// TIA Portal V19 program export: 4 tag tables, 0 data types, 0 data blocks, 1 code blocks (in call order from the OBs), 0 instance data blocks

VAR_GLOBAL   // PLC tag table "conveyor-0"
   "Start Button 0" AT %I0.0 : Bool;
   "Belt Conveyor (4m) 0" AT %Q0.0 : Bool;
   "memedge0-0" AT %M0.0 : Bool;
   "memedge0-1" AT %M0.1 : Bool;
   "memedge0-2" AT %M0.2 : Bool;
   "mem0-start" AT %M0.3 : Bool;
   "memory0-0" AT %M0.4 : Bool;
   "memedge0-3" AT %M0.5 : Bool;
   "memedge0-4" AT %M0.6 : Bool;
   "memedge0-5" AT %M0.7 : Bool;
END_VAR

VAR_GLOBAL   // PLC tag table "conveyor-1"
   "Start Button 1" AT %I0.1 : Bool;
   "Stop Button 1" AT %I0.2 : Bool;
   "Belt Conveyor (4m) 1" AT %Q0.1 : Bool;
END_VAR

VAR_GLOBAL   // PLC tag table "conveyor-2"
   "Start Button 2-Left" AT %I0.3 : Bool;
   "Start Button 2-right" AT %I0.4 : Bool;
   "Stop Button 2" AT %I0.5 : Bool;
   "Belt Conveyor (4m) 2 (+)" AT %Q0.2 : Bool;
   "Belt Conveyor (4m) 2 (-)" AT %Q0.3 : Bool;
   "mem2-start-right" AT %M2.0 : Bool;
   "mem2-start-left" AT %M2.1 : Bool;
   "mem2-stop" AT %M2.2 : Bool;
   "mem-Belt Conveyor (4m) 2 (+)" AT %M2.3 : Bool;
   "mem-Belt Conveyor (4m) 2 (-)" AT %M2.4 : Bool;
   "mem-moment" AT %M2.5 : Bool;
END_VAR

VAR_GLOBAL   // PLC tag table "conveyor6m"
   "Belt Conveyor (6m) 0" AT %Q0.4 : Bool;
   "memedge-6m-0" AT %M1.0 : Bool;
   "memedge-6m-1" AT %M1.1 : Bool;
   "memedge-6m-2" AT %M1.2 : Bool;
   "memedge-6m-3" AT %M1.3 : Bool;
   "memedge-6m-4" AT %M1.4 : Bool;
   "memedge-6m-5" AT %M1.5 : Bool;
   "mem-6m-start" AT %M1.6 : Bool;
   "memory-6m-0" AT %M1.7 : Bool;
END_VAR

ORGANIZATION_BLOCK "Main"   // OB1, LAD, ProgramCycle
TITLE = "Main Program Sweep (Cycle)"
{ S7_Optimized_Access := 'TRUE' }
// stored: SetENOAutomatically false
   VAR_INPUT
      Initial_Call : Bool;   // Initial call of this OB
      Remanence : Bool;   // =True, if remanent data are available
   END_VAR
   VAR_TEMP   // added for the SCL form of the ladder/FBD networks
      _w1 : Bool;
      _w2 : Bool;
   END_VAR
BEGIN

REGION Network 1: start and stop with one button ( physical & scada)
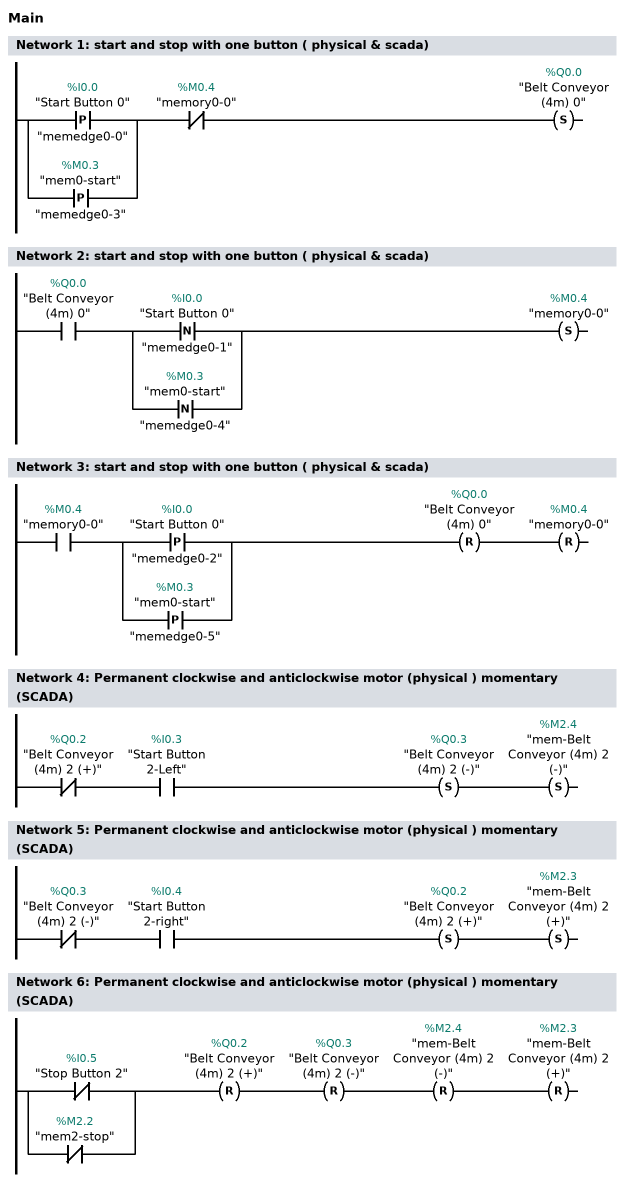
   RUNG wire#powerrail
      P_Contact(operand := "Start Button 0", bit := "memedge0-0")
      wire#w1
      I_Contact( "memory0-0" )
      S_Coil( "Belt Conveyor (4m) 0" )
   END_RUNG
   RUNG wire#powerrail
      P_Contact(operand := "mem0-start", bit := "memedge0-3")
   END_RUNG wire#w1
   // the same network as SCL:
   #_w1 := "Start Button 0" AND NOT "memedge0-0";   // rising edge of "Start Button 0"
   "memedge0-0" := "Start Button 0";
   #_w2 := "mem0-start" AND NOT "memedge0-3";   // rising edge of "mem0-start"
   "memedge0-3" := "mem0-start";
   IF (#_w1 OR #_w2) AND NOT "memory0-0" THEN "Belt Conveyor (4m) 0" := TRUE; END_IF;
END_REGION

REGION Network 2: start and stop with one button ( physical & scada)
   RUNG wire#powerrail
      Contact( "Belt Conveyor (4m) 0" )
      wire#w1
      N_Contact(operand := "Start Button 0", bit := "memedge0-1")
      wire#w2
      S_Coil( "memory0-0" )
   END_RUNG
   RUNG wire#w1
      N_Contact(operand := "mem0-start", bit := "memedge0-4")
   END_RUNG wire#w2
   // the same network as SCL:
   #_w1 := "Belt Conveyor (4m) 0" AND NOT "Start Button 0" AND "memedge0-1";   // falling edge of "Start Button 0"
   "memedge0-1" := "Start Button 0";
   #_w2 := "Belt Conveyor (4m) 0" AND NOT "mem0-start" AND "memedge0-4";   // falling edge of "mem0-start"
   "memedge0-4" := "mem0-start";
   IF #_w1 OR #_w2 THEN "memory0-0" := TRUE; END_IF;
END_REGION

REGION Network 3: start and stop with one button ( physical & scada)
   RUNG wire#powerrail
      Contact( "memory0-0" )
      wire#w1
      P_Contact(operand := "Start Button 0", bit := "memedge0-2")
      wire#w2
      R_Coil( "Belt Conveyor (4m) 0" )
      R_Coil( "memory0-0" )
   END_RUNG
   RUNG wire#w1
      P_Contact(operand := "mem0-start", bit := "memedge0-5")
   END_RUNG wire#w2
   // the same network as SCL:
   #_w1 := "memory0-0" AND "Start Button 0" AND NOT "memedge0-2";   // rising edge of "Start Button 0"
   "memedge0-2" := "Start Button 0";
   #_w2 := "memory0-0" AND "mem0-start" AND NOT "memedge0-5";   // rising edge of "mem0-start"
   "memedge0-5" := "mem0-start";
   IF #_w1 OR #_w2 THEN
       "Belt Conveyor (4m) 0" := FALSE;
       "memory0-0" := FALSE;
   END_IF;
END_REGION

REGION Network 4: Permanent clockwise and anticlockwise motor (physical ) momentary (SCADA)
   RUNG wire#powerrail
      I_Contact( "Belt Conveyor (4m) 2 (+)" )
      Contact( "Start Button 2-Left" )
      S_Coil( "Belt Conveyor (4m) 2 (-)" )
      S_Coil( "mem-Belt Conveyor (4m) 2 (-)" )
   END_RUNG
   // the same network as SCL:
   IF NOT "Belt Conveyor (4m) 2 (+)" AND "Start Button 2-Left" THEN
       "Belt Conveyor (4m) 2 (-)" := TRUE;
       "mem-Belt Conveyor (4m) 2 (-)" := TRUE;
   END_IF;
END_REGION

REGION Network 5: Permanent clockwise and anticlockwise motor (physical ) momentary (SCADA)
   RUNG wire#powerrail
      I_Contact( "Belt Conveyor (4m) 2 (-)" )
      Contact( "Start Button 2-right" )
      S_Coil( "Belt Conveyor (4m) 2 (+)" )
      S_Coil( "mem-Belt Conveyor (4m) 2 (+)" )
   END_RUNG
   // the same network as SCL:
   IF NOT "Belt Conveyor (4m) 2 (-)" AND "Start Button 2-right" THEN
       "Belt Conveyor (4m) 2 (+)" := TRUE;
       "mem-Belt Conveyor (4m) 2 (+)" := TRUE;
   END_IF;
END_REGION

REGION Network 6: Permanent clockwise and anticlockwise motor (physical ) momentary (SCADA)
   RUNG wire#powerrail
      I_Contact( "Stop Button 2" )
      wire#w1
      R_Coil( "Belt Conveyor (4m) 2 (+)" )
      R_Coil( "Belt Conveyor (4m) 2 (-)" )
      R_Coil( "mem-Belt Conveyor (4m) 2 (-)" )
      R_Coil( "mem-Belt Conveyor (4m) 2 (+)" )
   END_RUNG
   RUNG wire#powerrail
      I_Contact( "mem2-stop" )
   END_RUNG wire#w1
   // the same network as SCL:
   IF NOT "Stop Button 2" OR NOT "mem2-stop" THEN
       "Belt Conveyor (4m) 2 (+)" := FALSE;
       "Belt Conveyor (4m) 2 (-)" := FALSE;
       "mem-Belt Conveyor (4m) 2 (-)" := FALSE;
       "mem-Belt Conveyor (4m) 2 (+)" := FALSE;
   END_IF;
END_REGION
END_ORGANIZATION_BLOCK
